FUNCTION_BLOCK "FbSum1bit"
TITLE = 'Сумматор 1бит.'

{ S7_read_back := 'true' ;
  S7_blockview := 'big'  }

AUTHOR  : VA
FAMILY  : LIB_PLC
VERSION : '1.0'

VAR_INPUT // Входные переменные.
A   :BOOL := FALSE; // Первое слагаемое.
B   :BOOL := FALSE; // Второе слагаемое.
Cin :BOOL := FALSE; // Входной флаг переноса при сложении.
END_VAR

VAR_OUTPUT // Выходные переменные.
Sum  :BOOL := FALSE; // Сумма.
Cout :BOOL := FALSE; // Выходной флаг переноса при сложении.
END_VAR

BEGIN

// Сумма.
Sum := (NOT(A) AND NOT(B) AND Cin) OR (NOT(A) AND B AND NOT(Cin)) OR (A AND NOT(B) AND NOT(Cin)) OR (A AND B AND Cin);
// Перенос.
Cout := (NOT(A) AND B AND Cin) OR (A AND NOT(B) AND Cin) OR (A AND B AND NOT(Cin)) OR (A AND B AND Cin);

// Таблица истинности сумматора.
// +---+---+-----+-----+------+
// | A | B | Cin | Sum | Cout |
// +---+---+-----+-----+------+
// | 0 | 0 | 0   | 0   | 0    |
// +---+---+-----+-----+------+
// | 0 | 0 | 1   | 1   | 0    |
// +---+---+-----+-----+------+
// | 0 | 1 | 0   | 1   | 0    |
// +---+---+-----+-----+------+
// | 0 | 1 | 1   | 0   | 1    |
// +---+---+-----+-----+------+
// | 1 | 0 | 0   | 1   | 0    |
// +---+---+-----+-----+------+
// | 1 | 0 | 1   | 0   | 1    |
// +---+---+-----+-----+------+
// | 1 | 1 | 0   | 0   | 1    |
// +---+---+-----+-----+------+
// | 1 | 1 | 1   | 1   | 1    |
// +---+---+-----+-----+------+
// Получившийся сумматор состоит из 31ой элементарной операций типа И,ИЛИ,НЕ.
// Данная реализация самая наглядная но не факт, что оптимальная.
// Сумма формируется 4мя дешифраторами соединенными по схеме ИЛИ.
// Флаг переноса формируется 4мя дешифраторами соединенными по схеме ИЛИ.
// Сумматор подходит для целых 8битных чисел без знаком 0...255. (тестировано.)
// Сумматор подходит для целых 7битных чисел со знаком -127...127. (надо протестировать заем...)

//********************************************************

// AND
// |    X1       X2       Y1   |
// +---| |------| |------( )---+
// |                           |

// OR
// |    X1           Y1   |
// +---| |---+------( )---+
// |         |            |
// |    X2   |            |
// +---| |---+            |
// |                      |

// NOT
// |    X1       Y1   |
// +---|/|------( )---+
// |                  |

//********************************************************

//        +-----+   +-----+   +----+
//   A ->-| NOT |->-| AND |->-| OR |->- Sum
//        +-----+   |     |   |    |
//        +-----+   |     |   |    |
//   B ->-| NOT |->-|     |   |    |
//        +-----+   |     |   |    |
//                  |     |   |    |
// Cin ->-----------|     |   |    |
//                  +-----+   |    |
//        +-----+   +-----+   |    |
//   A ->-| NOT |->-| AND |->-|    |
//        +-----+   |     |   |    |
//                  |     |   |    |
//   B ->-----------|     |   |    |
//                  |     |   |    |
//        +-----+   |     |   |    |
// Cin ->-| NOT |->-|     |   |    |
//        +-----+   +-----+   |    |
//                  +-----+   |    |
//   A ->-----------| AND |->-|    |
//                  |     |   |    |
//        +-----+   |     |   |    |
//   B ->-| NOT |->-|     |   |    |
//        +-----+   |     |   |    |
//        +-----+   |     |   |    |
// Cin ->-| NOT |->-|     |   |    |
//        +-----+   +-----+   |    |
//                  +-----+   |    |
//   A ->-----------| AND |   |    |
//                  |     |   |    |
//                  |     |   |    |
//   B ->-----------|     |   |    |
//                  |     |   |    |
//                  |     |   |    |
// Cin ->-----------|     |   |    |
//                  +-----+   +----+

//    +--------+
// ->-|Cin  Sum|->-
// ->-|A       |
// ->-|B       |
//    +--------+

//        +-----+   +-----+   +----+
//   A ->-| NOT |->-| AND |->-| OR |->- Cout
//        +-----+   |     |   |    |
//                  |     |   |    |
//   B ->-----------|     |   |    |
//                  |     |   |    |
//                  |     |   |    |
// Cin ->-----------|     |   |    |
//                  +-----+   |    |
//                  +-----+   |    |
//   A ->-----------| AND |->-|    |
//                  |     |   |    |
//        +-----+   |     |   |    |
//   B ->-| NOT |->-|     |   |    |
//        +-----+   |     |   |    |
//                  |     |   |    |
// Cin ->-----------|     |   |    |
//                  +-----+   |    |
//                  +-----+   |    |
//   A ->-----------| AND |->-|    |
//                  |     |   |    |
//                  |     |   |    |
//   B ->-----------|     |   |    |
//                  |     |   |    |
//        +-----+   |     |   |    |
// Cin ->-| NOT |->-|     |   |    |
//        +-----+   +-----+   |    |
//                  +-----+   |    |
//   A ->-----------| AND |->-|    |
//                  |     |   |    |
//                  |     |   |    |
//   B ->-----------|     |   |    |
//                  |     |   |    |
//                  |     |   |    |
// Cin ->-----------|     |   |    |
//                  +-----+   +----+

//    +--------+
// ->-|Cin Cout|->-
// ->-|A       |
// ->-|B       |
//    +--------+

//********************************************************

//       +--------+
//  0 ->-|Cin  Sum|->- Sum0
// A0 ->-|A   Cout|->-+
// B0 ->-|B       |   |
//       +--------+   |
//                    |
//   +----------------+
//   |
//   |   +--------+
//   +->-|Cin  Sum|->- Sum1
// A1 ->-|A   Cout|->-+
// B1 ->-|B       |   |
//       +--------+   |
//                    |
//   +----------------+
//   |
//   |   +--------+
//   +->-|Cin  Sum|->- Sum2
// A2 ->-|A   Cout|->-+
// B2 ->-|B       |   |
//       +--------+   |
//                    |
//   +----------------+
//   |
//   |   +--------+
//   +->-|Cin  Sum|->- Sum3
// A3 ->-|A   Cout|->-+
// B3 ->-|B       |   |
//       +--------+   |
//                    |
//   +----------------+
//   |
//   |   +--------+
//   +->-|Cin  Sum|->- Sum4
// A4 ->-|A   Cout|->-+
// B4 ->-|B       |   |
//       +--------+   |
//                    |
//   +----------------+
//   |
//   |   +--------+
//   +->-|Cin  Sum|->- Sum5
// A5 ->-|A   Cout|->-+
// B5 ->-|B       |   |
//       +--------+   |
//                    |
//   +----------------+
//   |
//   |   +--------+
//   +->-|Cin  Sum|->- Sum6
// A6 ->-|A   Cout|->-+
// B6 ->-|B       |   |
//       +--------+   |
//                    |
//   +----------------+
//   |
//   |   +--------+
//   +->-|Cin  Sum|->- Sum7
// A7 ->-|A   Cout|->- Cout
// B7 ->-|B       |
//       +--------+

//********************************************************

// AVR ASM
// LDI R16,2
// LDI R17,3
// ADD R16, R17

//********************************************************

// GCC
// uint8_t add(uint8_t A, uint8_t B) {
// return (A + B); }

//********************************************************

// @COPYLEFT ALL WRONGS RESERVED :)
// Author: VA
// Contacts: DIY.PLC.314@gmail.com
// Date start LIB_PLC: 2014
// License: GNU GPL-2.0-or-later
// https://www.gnu.org/licenses/old-licenses/gpl-2.0.html
// https://www.youtube.com/watch?v=n1F_MfLRlX0
// https://www.youtube.com/@DIY_PLC
// https://github.com/DIYPLC/LIB_PLC
// https://oshwlab.com/diy.plc.314/PLC_HW1_SW1
// https://3dtoday.ru/3d-models/mechanical-parts/body/korpus-na-din-reiku
// https://t.me/DIY_PLC
// https://drive.google.com/drive/folders/16GDX0i07rwDrl_oPzL-lQAqMiAz3ouJV?usp=sharing

END_FUNCTION_BLOCK
